Fanuc TP program (LS listing): _boot.ls

/PROG  _BOOT
/ATTR
OWNER		= MNEDITOR;
COMMENT		= "";
PROG_SIZE	= 199;
CREATE		= DATE 00-01-04  TIME 22:36:00;
MODIFIED	= DATE 23-05-03  TIME 12:19:18;
FILE_NAME	= ;
VERSION		= 0;
LINE_COUNT	= 2;
MEMORY_SIZE	= 571;
PROTECT		= READ_WRITE;
TCD:  STACK_SIZE	= 0,
      TASK_PRIORITY	= 50,
      TIME_SLICE	= 0,
      BUSY_LAMP_OFF	= 0,
      ABORT_REQUEST	= 0,
      PAUSE_REQUEST	= 0;
DEFAULT_GROUP	= *,*,*,*,*;
CONTROL_CODE	= 00000000 00000000;
LOCAL_REGISTERS	= 0,0,0;
/APPL
/APPL

AUTO_SINGULARITY_HEADER;
  ENABLE_SINGULARITY_AVOIDANCE   : FALSE;
/MN
   1:  WAIT  10.00(sec) ;
   2:  RUN _BGT_STARTUP ;
/POS
/END
